(* CoDeSys 2.3.9.29 project: test2.pro *)
(* Libraries: STANDARD.LIB 4.10.05 11:14:46, IECSFC.LIB 13.4.06 15:51:28, SYSLIBTIME.LIB 20.2.06 13:31:16, SYSTASKINFO.LIB 20.2.06 13:31:38, ANALYZATION.LIB 5.10.99 09:05:06, SYSLIBCALLBACK.LIB 20.2.06 13:31:08 *)

(* PLC configuration (modules and I/O channels)
Discrete input 8 bit [ID100] node 0, in %IB0 out %QB0 {Filtrationtime = 10; Filtrationtime = 10; Filtrationtime = 10; Filtrationtime = 10; Filtrationtime = 10; Filtrationtime = 10; Filtrationtime = 10; Filtrationtime = 10; Visibility = No; PinCount = 8; WatchDogPeriod = 1000; PollPeriod = 1}
  AT %IB0.0 [ByteInput] 8 discrete inputs
Discrete output 2 bit [ID101] node 1, in %IB1 out %QB1 {PinCount = 2; SafeValueBool = FALSE; SafeValueBool = FALSE; Visibility = No}
  AT %QX1.0 [BitOutput] First
  AT %QX1.1 [BitOutput] Second
Discrete output 2 bit [ID101] node 2, in %IB2 out %QB2 {PinCount = 2; SafeValueBool = FALSE; SafeValueBool = FALSE; Visibility = No}
  AT %QX2.0 [BitOutput] First
  AT %QX2.1 [BitOutput] Second
Discrete output 2 bit [ID101] node 3, in %IB3 out %QB3 {PinCount = 2; SafeValueBool = FALSE; SafeValueBool = FALSE; Visibility = No}
  AT %QX3.0 [BitOutput] First
  AT %QX3.1 [BitOutput] Second
Discrete output 2 bit [ID101] node 4, in %IB4 out %QB4 {PinCount = 2; SafeValueBool = FALSE; SafeValueBool = FALSE; Visibility = No}
  AT %QX4.0 [BitOutput] First
  AT %QX4.1 [BitOutput] Second
Discrete output 2 bit [ID101] node 5, in %IB5 out %QB5 {PinCount = 2; SafeValueBool = FALSE; SafeValueBool = FALSE; Visibility = No}
  AT %QX5.0 [BitOutput] First
  AT %QX5.1 [BitOutput] Second
Discrete output 2 bit [ID101] node 6, in %IB6 out %QB6 {PinCount = 2; SafeValueBool = FALSE; SafeValueBool = FALSE; Visibility = No}
  AT %QX6.0 [BitOutput] First
  AT %QX6.1 [BitOutput] Second
Special output [ID104] node 7, in %IB7 out %QB7 {Visibility = No; PinCount = 1}
  AT %QX7.0 [BitOutput] Special output
TCP [TCP_ID221] node 0, in %IB8.0.0 out %QB8.0.0 {RemotePort = 502; Visibility = No}
x001 AT %QB8.1.0 [ByteOutput]
x002 AT %QD8.2.0 [DWordOutput]
x003 AT %QW8.3.0 [WordOutput]
x004 AT %QD8.4.0 [DWordOutput]
x005 AT %QB8.5.0 [ByteOutput]
x006 AT %QB8.6.0 [ByteOutput]
x007 AT %QD8.7.0 [FloatOutput]
*)

(* Global variable list: Global_Variables *)
VAR_GLOBAL
	_tm: DWORD;
END_VAR

(* POU PLC_PRG, ST *)
PROGRAM PLC_PRG
VAR
	tm: DWORD;
END_VAR
tm:=TIME_TO_DWORD(TIME());
IF tm-_tm>=1000 THEN
	_tm:=tm;
	x002:=x002+x001;
	x003:=x003+x005;
	x004:=x004+x006;
	x007:=x007+0.0001;
END_IF
END_PROGRAM
